FUNCTION FC_Durchschnitt : REAL				// FC um Durchschnitt zu berechnen
VAR_INPUT
	vii_Wert_1 : INT;						// Einganswert 1
	vii_Wert_2 : INT;						// Einganswert 2
	vii_Wert_3 : INT;						// Einganswert 3
END_VAR
VAR_OUTPUT
END_VAR
VAR
END_VAR

 FC_Durchschnitt := INT_TO_REAL(vii_Wert_1 + vii_Wert_2 + vii_Wert_3) / 3;			// Addition der 3 Werte anschliessend :3 um den Schnitt zu erhalten
// Funktion kann, mit der Übergabe 3er Werte, aus einem beliebigen FB aufgerufen werden. Auch als Multiinstanz aufrufbar

END_FUNCTION

(* stored: Version 1.1.0.1
   POU FC_Durchschnitt: Id {5fd35583-b519-4c4c-9016-ca68ce2edbce}, SpecialFunc None *)
